(* PLC project graf, TNI-Software ControlBuild 4.00 *)
(* stored: creationDateTime 2018-09-17T17:24:47-01:00 *)

(* CB.Or_Divergences_Exclusivity=true *)
FUNCTION_BLOCK tapis_conv.graf
  VAR_INPUT  (* CB.group=Retour_PO CB.kind=inputVars *)
    Fin_Convoyage : BOOL := false;
  END_VAR
  VAR_INPUT  (* CB.group=Retour_Utilisateur CB.kind=inputVars *)
    Chargement : BOOL := false;
    Dechargement : BOOL := false;
  END_VAR
  VAR_OUTPUT  (* CB.group=Commande_PO CB.kind=outputVars *)
    Marche : BOOL := false;
  END_VAR
  VAR  (* CB.kind=localVars *)
    nb_piece : DINT := 0;
  END_VAR

INITIAL_STEP 10:
  COMPUTE_FUNCTION_BLOCKS(S);
END_STEP
TRANSITION FROM 10 TO 11
  := Chargement and nb_piece<10;
END_TRANSITION
INITIAL_STEP 20:
END_STEP
TRANSITION FROM 20 TO 21
  := Dechargement and nb_piece>0;
END_TRANSITION
STEP 21:
  21_INLINE1(N);
END_STEP
ACTION 21_INLINE1:
  nb_piece:=nb_piece-1;
END_ACTION
TRANSITION FROM 21 TO 20
  := TRUE;
END_TRANSITION
STEP 11:
  11_INLINE2(N);
END_STEP
ACTION 11_INLINE2:
  Marche;
  nb_piece:=nb_piece+1;
END_ACTION
TRANSITION FROM 11 TO 10
  := Fin_Convoyage;
END_TRANSITION
ACTION COMPUTE_FUNCTION_BLOCKS:  (* blocks drawn on the SFC sheet *)
  G1:
  G2:
END_ACTION
END_FUNCTION_BLOCK
